DATA_BLOCK "A0301_Fermi_P2"   // DB36
// stored: InstanceOfName A0301_Fermi_P2_FB, InstanceOfType FB
"A0301_Fermi_P2_FB"
BEGIN
   AreaInterface.EStop := FALSE;
   AreaInterface.Man := TRUE;
   AreaInterface.Aut := FALSE;
   AreaInterface.Cycle := FALSE;
   AreaInterface.StopInPhase := FALSE;
   AreaInterface.StopProgrammed := FALSE;
   AreaInterface.RstAlarms := FALSE;
   AreaInterface.ManOneShot := FALSE;
   AreaInterface.AutOneShot := FALSE;
   AreaInterface.CycleOneShot := FALSE;
   AreaInterface.CheckAutReady := FALSE;
   ZSI.Door_NormalStop := FALSE;
   ZSI.Door_SafeStop := FALSE;
   ZSI.Door_Opened := FALSE;
   ZSI.Door_EntryEnable := FALSE;
   DSI.SafeStop := FALSE;
   DSI.PowerEnable := TRUE;
   DSI.DevicesInSafeState := FALSE;
   CIn.Manager_Fermi.EnableStopDoorOpeningReq := FALSE;
   CIn.Manager_Fermi.EnableStopInPhase := FALSE;
   CIn.Manager_Fermi.EnableStopProgrammed := FALSE;
   CIn.Manager_Fermi.Control_ON := FALSE;
   CIn.Manager_Fermi.Rest := FALSE;
   CIn.Manager_Fermi.Work := FALSE;
   CIn.P1.Fermi.CtrlSafe := FALSE;
   CIn.P1.Fermi.Standstill := TRUE;
   CIn.P1.Fermi.ReqOilPressure := FALSE;
   CIn.P1.Fermi.Rest_CheckNext := FALSE;
   CIn.P1.Fermi.Work_CheckNext := FALSE;
   CIn.P1.Fermi.Rest := FALSE;
   CIn.P1.Fermi.Work := FALSE;
   CIn.P1.Pareggiatore.CtrlSafe := FALSE;
   CIn.P1.Pareggiatore.Standstill := TRUE;
   CIn.P1.Pareggiatore.ReqOilPressure := FALSE;
   CIn.P1.Pareggiatore.Rest_CheckNext := FALSE;
   CIn.P1.Pareggiatore.Work_CheckNext := FALSE;
   CIn.P1.Pareggiatore.Rest := FALSE;
   CIn.P1.Pareggiatore.Work := FALSE;
   CIn.Trasporto.Infeed_ReqON := FALSE;
   CIn.Trasporto.CtrlSafe := FALSE;
   CIn.Trasporto.Standstill := TRUE;
   CIn.Trasporto.Bwd_CheckNext := FALSE;
   CIn.Trasporto.Fwd_CheckNext := FALSE;
   CIn.Trasporto.Bwd_VelZero := FALSE;
   CIn.Trasporto.Bwd_Running := FALSE;
   CIn.Trasporto.Fwd_VelZero := FALSE;
   CIn.Trasporto.Fwd_Running := FALSE;
   CIn.Trasporto.ActualVelocity := 0.0;
   CIn.Trasporto.TargetVelocity := 0.0;
   CIn.Trasporto.MaxVelocity := 39597.8;
   Config.Fermi[1..6].DelayPressureRunningTimeout := T#3S;
   Config.Fermi[1..6].DelayMissingCondition := T#3S;
   Config.Fermi[1..6].Rest_LsQty := 1;
   Config.Fermi[1..6].Work_LsQty := 0;
   Config.Fermi[1..6].Rest_RetainAut := FALSE;
   Config.Fermi[1..6].Work_RetainAut := FALSE;
   Config.Fermi[1..6].V.RestLimSwitchExist := TRUE;
   Config.Fermi[1..6].V.WorkLimSwitchExist := FALSE;
   Config.Fermi[1..6].V.CheckOilInPressure := FALSE;
   Config.Fermi[1..6].V.CutRestWhenIsAtRest := TRUE;
   Config.Fermi[1..6].V.CutWorkWhenIsAtWork := TRUE;
   Config.Fermi[1..6].V.RestTime := T#2S;
   Config.Fermi[1..6].V.WorkTime := T#2S;
   Config.Fermi[1..6].V.RestTimeOut := T#1H;
   Config.Fermi[1..6].V.WorkTimeOut := T#1H;
   Config.Sollevatori[1..6].DelayPressureRunningTimeout := T#3S;
   Config.Sollevatori[1..6].DelayMissingCondition := T#3S;
   Config.Sollevatori[1..6].Rest_LsQty := 1;
   Config.Sollevatori[1..6].Work_LsQty := 0;
   Config.Sollevatori[1..6].Rest_RetainAut := FALSE;
   Config.Sollevatori[1..6].Work_RetainAut := FALSE;
   Config.Sollevatori[1..6].V.RestLimSwitchExist := TRUE;
   Config.Sollevatori[1..6].V.WorkLimSwitchExist := FALSE;
   Config.Sollevatori[1..6].V.CheckOilInPressure := FALSE;
   Config.Sollevatori[1..6].V.CutRestWhenIsAtRest := TRUE;
   Config.Sollevatori[1..6].V.CutWorkWhenIsAtWork := TRUE;
   Config.Sollevatori[1..6].V.RestTime := T#2S;
   Config.Sollevatori[1..6].V.WorkTime := T#2S;
   Config.Sollevatori[1..6].V.RestTimeOut := T#1H;
   Config.Sollevatori[1..6].V.WorkTimeOut := T#1H;
   MachineInterface.AutReady := FALSE;
   MachineInterface.Aborting := FALSE;
   MachineInterface.AckStopInPhase := FALSE;
   MachineInterface.AckStopProgrammed := FALSE;
   MachineInterface.MotionsStandStill := TRUE;
   MachineInterface.AlarmsPresence := FALSE;
   MachineInterface.WarningPresence := FALSE;
   COut.Fermi.CtrlSafe := FALSE;
   COut.Fermi.Standstill := TRUE;
   COut.Fermi.ReqOilPressure := FALSE;
   COut.Fermi.Rest_CheckNext := FALSE;
   COut.Fermi.Work_CheckNext := FALSE;
   COut.Fermi.Rest := FALSE;
   COut.Fermi.Work := FALSE;
   COut.Sollevatori.CtrlSafe := FALSE;
   COut.Sollevatori.Standstill := TRUE;
   COut.Sollevatori.ReqOilPressure := FALSE;
   COut.Sollevatori.Rest_CheckNext := FALSE;
   COut.Sollevatori.Work_CheckNext := FALSE;
   COut.Sollevatori.Rest := FALSE;
   COut.Sollevatori.Work := FALSE;
   Alarm.Fermi[1..6].TimeOutRest := FALSE;
   Alarm.Fermi[1..6].TimeOutWork := FALSE;
   Alarm.Fermi[1..6].LimitSwitches := FALSE;
   Alarm.Sollevatori[1..6].TimeOutRest := FALSE;
   Alarm.Sollevatori[1..6].TimeOutWork := FALSE;
   Alarm.Sollevatori[1..6].LimitSwitches := FALSE;
   Warning.Fermi[1..6].NotAutReady := FALSE;
   Warning.Fermi[1..6].PressureRunning_Timeout := FALSE;
   Warning.Fermi[1..6].Rest_MissingExtEnable := FALSE;
   Warning.Fermi[1..6].Work_MissingExtEnable := FALSE;
   Warning.Fermi[1].Missing_Rest_Ls_ON[1..8] := FALSE;
   Warning.Fermi[2].Missing_Rest_Ls_ON[1..8] := FALSE;
   Warning.Fermi[3].Missing_Rest_Ls_ON[1..8] := FALSE;
   Warning.Fermi[4].Missing_Rest_Ls_ON[1..8] := FALSE;
   Warning.Fermi[5].Missing_Rest_Ls_ON[1..8] := FALSE;
   Warning.Fermi[6].Missing_Rest_Ls_ON[1..8] := FALSE;
   Warning.Fermi[1].Missing_Work_Ls_ON[1..8] := FALSE;
   Warning.Fermi[2].Missing_Work_Ls_ON[1..8] := FALSE;
   Warning.Fermi[3].Missing_Work_Ls_ON[1..8] := FALSE;
   Warning.Fermi[4].Missing_Work_Ls_ON[1..8] := FALSE;
   Warning.Fermi[5].Missing_Work_Ls_ON[1..8] := FALSE;
   Warning.Fermi[6].Missing_Work_Ls_ON[1..8] := FALSE;
   Warning.Sollevatori[1..6].NotAutReady := FALSE;
   Warning.Sollevatori[1..6].PressureRunning_Timeout := FALSE;
   Warning.Sollevatori[1..6].Rest_MissingExtEnable := FALSE;
   Warning.Sollevatori[1..6].Work_MissingExtEnable := FALSE;
   Warning.Sollevatori[1].Missing_Rest_Ls_ON[1..8] := FALSE;
   Warning.Sollevatori[2].Missing_Rest_Ls_ON[1..8] := FALSE;
   Warning.Sollevatori[3].Missing_Rest_Ls_ON[1..8] := FALSE;
   Warning.Sollevatori[4].Missing_Rest_Ls_ON[1..8] := FALSE;
   Warning.Sollevatori[5].Missing_Rest_Ls_ON[1..8] := FALSE;
   Warning.Sollevatori[6].Missing_Rest_Ls_ON[1..8] := FALSE;
   Warning.Sollevatori[1].Missing_Work_Ls_ON[1..8] := FALSE;
   Warning.Sollevatori[2].Missing_Work_Ls_ON[1..8] := FALSE;
   Warning.Sollevatori[3].Missing_Work_Ls_ON[1..8] := FALSE;
   Warning.Sollevatori[4].Missing_Work_Ls_ON[1..8] := FALSE;
   Warning.Sollevatori[5].Missing_Work_Ls_ON[1..8] := FALSE;
   Warning.Sollevatori[6].Missing_Work_Ls_ON[1..8] := FALSE;
   HMI.Selection[1..6] := TRUE;
   HMI.FermiSts.Standstill := TRUE;
   HMI.FermiSts.Rest := FALSE;
   HMI.FermiSts.Work := FALSE;
   HMI.FermiSts.AlarmPresence := FALSE;
   HMI.SollevatoriSts.Standstill := TRUE;
   HMI.SollevatoriSts.Rest := FALSE;
   HMI.SollevatoriSts.Work := FALSE;
   HMI.SollevatoriSts.AlarmPresence := FALSE;
   Fermi[1..6].AreaInterface.EStop := FALSE;
   Fermi[1..6].AreaInterface.Man := TRUE;
   Fermi[1..6].AreaInterface.Aut := FALSE;
   Fermi[1..6].AreaInterface.Cycle := FALSE;
   Fermi[1..6].AreaInterface.StopInPhase := FALSE;
   Fermi[1..6].AreaInterface.StopProgrammed := FALSE;
   Fermi[1..6].AreaInterface.RstAlarms := FALSE;
   Fermi[1..6].AreaInterface.ManOneShot := FALSE;
   Fermi[1..6].AreaInterface.AutOneShot := FALSE;
   Fermi[1..6].AreaInterface.CycleOneShot := FALSE;
   Fermi[1..6].AreaInterface.CheckAutReady := FALSE;
   Fermi[1..6].ZSI.Door_NormalStop := FALSE;
   Fermi[1..6].ZSI.Door_SafeStop := FALSE;
   Fermi[1..6].ZSI.Door_Opened := FALSE;
   Fermi[1..6].ZSI.Door_EntryEnable := FALSE;
   Fermi[1..6].DSI.SafeStop := FALSE;
   Fermi[1..6].DSI.PowerEnable := TRUE;
   Fermi[1..6].DSI.DevicesInSafeState := FALSE;
   Fermi[1..6].DataIn.PB.Rest := FALSE;
   Fermi[1..6].DataIn.PB.Work := FALSE;
   Fermi[1..6].DataIn.PB.StartStop := FALSE;
   Fermi[1].DataIn.Rest_Ls[1] := TRUE;
   Fermi[1].DataIn.Rest_Ls[2..8] := FALSE;
   Fermi[2].DataIn.Rest_Ls[1] := TRUE;
   Fermi[2].DataIn.Rest_Ls[2..8] := FALSE;
   Fermi[3].DataIn.Rest_Ls[1] := TRUE;
   Fermi[3].DataIn.Rest_Ls[2..8] := FALSE;
   Fermi[4].DataIn.Rest_Ls[1] := TRUE;
   Fermi[4].DataIn.Rest_Ls[2..8] := FALSE;
   Fermi[5].DataIn.Rest_Ls[1] := TRUE;
   Fermi[5].DataIn.Rest_Ls[2..8] := FALSE;
   Fermi[6].DataIn.Rest_Ls[1] := TRUE;
   Fermi[6].DataIn.Rest_Ls[2..8] := FALSE;
   Fermi[1].DataIn.Work_Ls[1..8] := FALSE;
   Fermi[2].DataIn.Work_Ls[1..8] := FALSE;
   Fermi[3].DataIn.Work_Ls[1..8] := FALSE;
   Fermi[4].DataIn.Work_Ls[1..8] := FALSE;
   Fermi[5].DataIn.Work_Ls[1..8] := FALSE;
   Fermi[6].DataIn.Work_Ls[1..8] := FALSE;
   Fermi[1..6].Cin.Manager.EnableStopDoorOpeningReq := FALSE;
   Fermi[1..6].Cin.Manager.EnableStopInPhase := FALSE;
   Fermi[1..6].Cin.Manager.EnableStopProgrammed := FALSE;
   Fermi[1..6].Cin.Manager.Control_ON := FALSE;
   Fermi[1..6].Cin.Manager.Rest := FALSE;
   Fermi[1..6].Cin.Manager.Work := FALSE;
   Fermi[1..6].Cin.PressureRunning := FALSE;
   Fermi[1..6].Cin.Rest_ExtEnable := TRUE;
   Fermi[1..6].Cin.Work_ExtEnable := TRUE;
   Fermi[1..6].Cin.ExternalAlarms := FALSE;
   Fermi[1..6].Config.DelayPressureRunningTimeout := T#3S;
   Fermi[1..6].Config.DelayMissingCondition := T#3S;
   Fermi[1..6].Config.Rest_LsQty := 1;
   Fermi[1..6].Config.Work_LsQty := 0;
   Fermi[1..6].Config.Rest_RetainAut := FALSE;
   Fermi[1..6].Config.Work_RetainAut := FALSE;
   Fermi[1..6].Config.V.RestLimSwitchExist := TRUE;
   Fermi[1..6].Config.V.WorkLimSwitchExist := FALSE;
   Fermi[1..6].Config.V.CheckOilInPressure := FALSE;
   Fermi[1..6].Config.V.CutRestWhenIsAtRest := TRUE;
   Fermi[1..6].Config.V.CutWorkWhenIsAtWork := TRUE;
   Fermi[1..6].Config.V.RestTime := T#2S;
   Fermi[1..6].Config.V.WorkTime := T#2S;
   Fermi[1..6].Config.V.RestTimeOut := T#1H;
   Fermi[1..6].Config.V.WorkTimeOut := T#1H;
   Fermi[1..6].MachineInterface.AutReady := FALSE;
   Fermi[1..6].MachineInterface.Aborting := FALSE;
   Fermi[1..6].MachineInterface.AckStopInPhase := FALSE;
   Fermi[1..6].MachineInterface.AckStopProgrammed := FALSE;
   Fermi[1..6].MachineInterface.MotionsStandStill := TRUE;
   Fermi[1..6].MachineInterface.AlarmsPresence := FALSE;
   Fermi[1..6].MachineInterface.WarningPresence := FALSE;
   Fermi[1..6].COut.CtrlSafe := FALSE;
   Fermi[1..6].COut.Standstill := TRUE;
   Fermi[1..6].COut.ReqOilPressure := FALSE;
   Fermi[1..6].COut.Rest_CheckNext := FALSE;
   Fermi[1..6].COut.Work_CheckNext := FALSE;
   Fermi[1..6].COut.Rest := TRUE;
   Fermi[1..6].COut.Work := FALSE;
   Fermi[1..6].DataOut.RestSolenoid := FALSE;
   Fermi[1..6].DataOut.WorkSolenoid := FALSE;
   Fermi[1..6].Sts.Standstill := TRUE;
   Fermi[1..6].Sts.AlarmsPresence := FALSE;
   Fermi[1..6].Sts.WarningsPresence := FALSE;
   Fermi[1..6].Sts.Rest_Cnd := TRUE;
   Fermi[1..6].Sts.Work_Cnd := TRUE;
   Fermi[1..6].Ctrl.StopDueDoorOpeningRequest := FALSE;
   Fermi[1..6].Ctrl.StopInPhase := FALSE;
   Fermi[1..6].Ctrl.StopProgrammed := FALSE;
   Fermi[1..6].Ctrl.StopAborting := FALSE;
   Fermi[1..6].Ctrl.Work := FALSE;
   Fermi[1..6].Ctrl.Rest := FALSE;
   Fermi[1..6].Ctrl.Rest_Man := FALSE;
   Fermi[1..6].Ctrl.Work_Man := FALSE;
   Fermi[1..6].Ctrl.Rest_Aut := FALSE;
   Fermi[1..6].Ctrl.Work_Aut := FALSE;
   Fermi[1..6].V.ValveCtrl.SafeStop := FALSE;
   Fermi[1..6].V.ValveCtrl.Rst := FALSE;
   Fermi[1..6].V.ValveCtrl.MoveRest := FALSE;
   Fermi[1..6].V.ValveCtrl.MoveWork := FALSE;
   Fermi[1..6].V.RestLimitSwitch := TRUE;
   Fermi[1..6].V.WorkLimitSwitch := FALSE;
   Fermi[1..6].V.OilInPressure := FALSE;
   Fermi[1..6].V.Simulation := FALSE;
   Fermi[1..6].V.Config.RestLimSwitchExist := TRUE;
   Fermi[1..6].V.Config.WorkLimSwitchExist := FALSE;
   Fermi[1..6].V.Config.CheckOilInPressure := FALSE;
   Fermi[1..6].V.Config.CutRestWhenIsAtRest := TRUE;
   Fermi[1..6].V.Config.CutWorkWhenIsAtWork := TRUE;
   Fermi[1..6].V.Config.RestTime := T#2S;
   Fermi[1..6].V.Config.WorkTime := T#2S;
   Fermi[1..6].V.Config.RestTimeOut := T#1H;
   Fermi[1..6].V.Config.WorkTimeOut := T#1H;
   Fermi[1..6].V.ValveSts.AlarmPresence := FALSE;
   Fermi[1..6].V.ValveSts.RestPermit := TRUE;
   Fermi[1..6].V.ValveSts.RestInProgress := FALSE;
   Fermi[1..6].V.ValveSts.IsAtRest := TRUE;
   Fermi[1..6].V.ValveSts.WorkPermit := TRUE;
   Fermi[1..6].V.ValveSts.WorkInProgress := FALSE;
   Fermi[1..6].V.ValveSts.IsAtWork := FALSE;
   Fermi[1..6].V.ValveSts.StandStill := TRUE;
   Fermi[1..6].V.RestSolenoid := FALSE;
   Fermi[1..6].V.WorkSolenoid := FALSE;
   Fermi[1..6].V.ReqOilPressure := FALSE;
   Fermi[1..6].V.IsAtRest := TRUE;
   Fermi[1..6].V.IsAtWork := FALSE;
   Fermi[1..6].V.Ctrl.RestReq := FALSE;
   Fermi[1..6].V.Ctrl.WorkReq := FALSE;
   Fermi[1..6].V.Ctrl.RestSolenoid := FALSE;
   Fermi[1..6].V.Ctrl.WorkSolenoid := FALSE;
   Fermi[1..6].V.tonRest.PT := T#2S;
   Fermi[1..6].V.tonRest.IN := TRUE;
   Fermi[1..6].V.tonWork.PT := T#0MS;
   Fermi[1..6].V.tonWork.IN := FALSE;
   Fermi[1..6].V.tonTimeOutRest.PT := T#0MS;
   Fermi[1..6].V.tonTimeOutRest.IN := FALSE;
   Fermi[1..6].V.tonTimeOutWork.PT := T#0MS;
   Fermi[1..6].V.tonTimeOutWork.IN := FALSE;
   Fermi[1..6].TON_NoPendingCmd.PT := T#500MS;
   Fermi[1..6].TON_NoPendingCmd.IN := TRUE;
   Fermi[1..6].TON_Rest_MissingExtEnable.PT := T#0MS;
   Fermi[1..6].TON_Rest_MissingExtEnable.IN := FALSE;
   Fermi[1..6].TON_Work_MissingExtEnable.PT := T#0MS;
   Fermi[1..6].TON_Work_MissingExtEnable.IN := FALSE;
   Fermi[1..6].TON_PressureRunning_Timeout.PT := T#0MS;
   Fermi[1..6].TON_PressureRunning_Timeout.IN := FALSE;
   Fermi[1..6].Aux.Pb_Rest := FALSE;
   Fermi[1..6].Aux.Pb_Work := FALSE;
   Fermi[1..6].Aux.Pb_StartStop := FALSE;
   Sollevatori[1..6].AreaInterface.EStop := FALSE;
   Sollevatori[1..6].AreaInterface.Man := TRUE;
   Sollevatori[1..6].AreaInterface.Aut := FALSE;
   Sollevatori[1..6].AreaInterface.Cycle := FALSE;
   Sollevatori[1..6].AreaInterface.StopInPhase := FALSE;
   Sollevatori[1..6].AreaInterface.StopProgrammed := FALSE;
   Sollevatori[1..6].AreaInterface.RstAlarms := FALSE;
   Sollevatori[1..6].AreaInterface.ManOneShot := FALSE;
   Sollevatori[1..6].AreaInterface.AutOneShot := FALSE;
   Sollevatori[1..6].AreaInterface.CycleOneShot := FALSE;
   Sollevatori[1..6].AreaInterface.CheckAutReady := FALSE;
   Sollevatori[1..6].ZSI.Door_NormalStop := FALSE;
   Sollevatori[1..6].ZSI.Door_SafeStop := FALSE;
   Sollevatori[1..6].ZSI.Door_Opened := FALSE;
   Sollevatori[1..6].ZSI.Door_EntryEnable := FALSE;
   Sollevatori[1..6].DSI.SafeStop := FALSE;
   Sollevatori[1..6].DSI.PowerEnable := TRUE;
   Sollevatori[1..6].DSI.DevicesInSafeState := FALSE;
   Sollevatori[1..6].DataIn.PB.Rest := FALSE;
   Sollevatori[1..6].DataIn.PB.Work := FALSE;
   Sollevatori[1..6].DataIn.PB.StartStop := FALSE;
   Sollevatori[1].DataIn.Rest_Ls[1] := TRUE;
   Sollevatori[1].DataIn.Rest_Ls[2..8] := FALSE;
   Sollevatori[2].DataIn.Rest_Ls[1] := TRUE;
   Sollevatori[2].DataIn.Rest_Ls[2..8] := FALSE;
   Sollevatori[3].DataIn.Rest_Ls[1] := TRUE;
   Sollevatori[3].DataIn.Rest_Ls[2..8] := FALSE;
   Sollevatori[4].DataIn.Rest_Ls[1] := TRUE;
   Sollevatori[4].DataIn.Rest_Ls[2..8] := FALSE;
   Sollevatori[5].DataIn.Rest_Ls[1] := TRUE;
   Sollevatori[5].DataIn.Rest_Ls[2..8] := FALSE;
   Sollevatori[6].DataIn.Rest_Ls[1] := TRUE;
   Sollevatori[6].DataIn.Rest_Ls[2..8] := FALSE;
   Sollevatori[1].DataIn.Work_Ls[1..8] := FALSE;
   Sollevatori[2].DataIn.Work_Ls[1..8] := FALSE;
   Sollevatori[3].DataIn.Work_Ls[1..8] := FALSE;
   Sollevatori[4].DataIn.Work_Ls[1..8] := FALSE;
   Sollevatori[5].DataIn.Work_Ls[1..8] := FALSE;
   Sollevatori[6].DataIn.Work_Ls[1..8] := FALSE;
   Sollevatori[1..6].Cin.Manager.EnableStopDoorOpeningReq := FALSE;
   Sollevatori[1..6].Cin.Manager.EnableStopInPhase := FALSE;
   Sollevatori[1..6].Cin.Manager.EnableStopProgrammed := FALSE;
   Sollevatori[1..6].Cin.Manager.Control_ON := FALSE;
   Sollevatori[1..6].Cin.Manager.Rest := FALSE;
   Sollevatori[1..6].Cin.Manager.Work := FALSE;
   Sollevatori[1..6].Cin.PressureRunning := FALSE;
   Sollevatori[1..6].Cin.Rest_ExtEnable := TRUE;
   Sollevatori[1..6].Cin.Work_ExtEnable := TRUE;
   Sollevatori[1..6].Cin.ExternalAlarms := FALSE;
   Sollevatori[1..6].Config.DelayPressureRunningTimeout := T#3S;
   Sollevatori[1..6].Config.DelayMissingCondition := T#3S;
   Sollevatori[1..6].Config.Rest_LsQty := 1;
   Sollevatori[1..6].Config.Work_LsQty := 0;
   Sollevatori[1..6].Config.Rest_RetainAut := FALSE;
   Sollevatori[1..6].Config.Work_RetainAut := FALSE;
   Sollevatori[1..6].Config.V.RestLimSwitchExist := TRUE;
   Sollevatori[1..6].Config.V.WorkLimSwitchExist := FALSE;
   Sollevatori[1..6].Config.V.CheckOilInPressure := FALSE;
   Sollevatori[1..6].Config.V.CutRestWhenIsAtRest := TRUE;
   Sollevatori[1..6].Config.V.CutWorkWhenIsAtWork := TRUE;
   Sollevatori[1..6].Config.V.RestTime := T#2S;
   Sollevatori[1..6].Config.V.WorkTime := T#2S;
   Sollevatori[1..6].Config.V.RestTimeOut := T#1H;
   Sollevatori[1..6].Config.V.WorkTimeOut := T#1H;
   Sollevatori[1..6].MachineInterface.AutReady := FALSE;
   Sollevatori[1..6].MachineInterface.Aborting := FALSE;
   Sollevatori[1..6].MachineInterface.AckStopInPhase := FALSE;
   Sollevatori[1..6].MachineInterface.AckStopProgrammed := FALSE;
   Sollevatori[1..6].MachineInterface.MotionsStandStill := TRUE;
   Sollevatori[1..6].MachineInterface.AlarmsPresence := FALSE;
   Sollevatori[1..6].MachineInterface.WarningPresence := FALSE;
   Sollevatori[1..6].COut.CtrlSafe := FALSE;
   Sollevatori[1..6].COut.Standstill := TRUE;
   Sollevatori[1..6].COut.ReqOilPressure := FALSE;
   Sollevatori[1..6].COut.Rest_CheckNext := FALSE;
   Sollevatori[1..6].COut.Work_CheckNext := FALSE;
   Sollevatori[1..6].COut.Rest := TRUE;
   Sollevatori[1..6].COut.Work := FALSE;
   Sollevatori[1..6].DataOut.RestSolenoid := FALSE;
   Sollevatori[1..6].DataOut.WorkSolenoid := FALSE;
   Sollevatori[1..6].Sts.Standstill := TRUE;
   Sollevatori[1..6].Sts.AlarmsPresence := FALSE;
   Sollevatori[1..6].Sts.WarningsPresence := FALSE;
   Sollevatori[1..6].Sts.Rest_Cnd := TRUE;
   Sollevatori[1..6].Sts.Work_Cnd := TRUE;
   Sollevatori[1..6].Ctrl.StopDueDoorOpeningRequest := FALSE;
   Sollevatori[1..6].Ctrl.StopInPhase := FALSE;
   Sollevatori[1..6].Ctrl.StopProgrammed := FALSE;
   Sollevatori[1..6].Ctrl.StopAborting := FALSE;
   Sollevatori[1..6].Ctrl.Work := FALSE;
   Sollevatori[1..6].Ctrl.Rest := FALSE;
   Sollevatori[1..6].Ctrl.Rest_Man := FALSE;
   Sollevatori[1..6].Ctrl.Work_Man := FALSE;
   Sollevatori[1..6].Ctrl.Rest_Aut := FALSE;
   Sollevatori[1..6].Ctrl.Work_Aut := FALSE;
   Sollevatori[1..6].V.ValveCtrl.SafeStop := FALSE;
   Sollevatori[1..6].V.ValveCtrl.Rst := FALSE;
   Sollevatori[1..6].V.ValveCtrl.MoveRest := FALSE;
   Sollevatori[1..6].V.ValveCtrl.MoveWork := FALSE;
   Sollevatori[1..6].V.RestLimitSwitch := TRUE;
   Sollevatori[1..6].V.WorkLimitSwitch := FALSE;
   Sollevatori[1..6].V.OilInPressure := FALSE;
   Sollevatori[1..6].V.Simulation := FALSE;
   Sollevatori[1..6].V.Config.RestLimSwitchExist := TRUE;
   Sollevatori[1..6].V.Config.WorkLimSwitchExist := FALSE;
   Sollevatori[1..6].V.Config.CheckOilInPressure := FALSE;
   Sollevatori[1..6].V.Config.CutRestWhenIsAtRest := TRUE;
   Sollevatori[1..6].V.Config.CutWorkWhenIsAtWork := TRUE;
   Sollevatori[1..6].V.Config.RestTime := T#2S;
   Sollevatori[1..6].V.Config.WorkTime := T#2S;
   Sollevatori[1..6].V.Config.RestTimeOut := T#1H;
   Sollevatori[1..6].V.Config.WorkTimeOut := T#1H;
   Sollevatori[1..6].V.ValveSts.AlarmPresence := FALSE;
   Sollevatori[1..6].V.ValveSts.RestPermit := TRUE;
   Sollevatori[1..6].V.ValveSts.RestInProgress := FALSE;
   Sollevatori[1..6].V.ValveSts.IsAtRest := TRUE;
   Sollevatori[1..6].V.ValveSts.WorkPermit := TRUE;
   Sollevatori[1..6].V.ValveSts.WorkInProgress := FALSE;
   Sollevatori[1..6].V.ValveSts.IsAtWork := FALSE;
   Sollevatori[1..6].V.ValveSts.StandStill := TRUE;
   Sollevatori[1..6].V.RestSolenoid := FALSE;
   Sollevatori[1..6].V.WorkSolenoid := FALSE;
   Sollevatori[1..6].V.ReqOilPressure := FALSE;
   Sollevatori[1..6].V.IsAtRest := TRUE;
   Sollevatori[1..6].V.IsAtWork := FALSE;
   Sollevatori[1..6].V.Ctrl.RestReq := FALSE;
   Sollevatori[1..6].V.Ctrl.WorkReq := FALSE;
   Sollevatori[1..6].V.Ctrl.RestSolenoid := FALSE;
   Sollevatori[1..6].V.Ctrl.WorkSolenoid := FALSE;
   Sollevatori[1..6].V.tonRest.PT := T#2S;
   Sollevatori[1..6].V.tonRest.IN := TRUE;
   Sollevatori[1..6].V.tonWork.PT := T#0MS;
   Sollevatori[1..6].V.tonWork.IN := FALSE;
   Sollevatori[1..6].V.tonTimeOutRest.PT := T#0MS;
   Sollevatori[1..6].V.tonTimeOutRest.IN := FALSE;
   Sollevatori[1..6].V.tonTimeOutWork.PT := T#0MS;
   Sollevatori[1..6].V.tonTimeOutWork.IN := FALSE;
   Sollevatori[1..6].TON_NoPendingCmd.PT := T#500MS;
   Sollevatori[1..6].TON_NoPendingCmd.IN := TRUE;
   Sollevatori[1..6].TON_Rest_MissingExtEnable.PT := T#0MS;
   Sollevatori[1..6].TON_Rest_MissingExtEnable.IN := FALSE;
   Sollevatori[1..6].TON_Work_MissingExtEnable.PT := T#0MS;
   Sollevatori[1..6].TON_Work_MissingExtEnable.IN := FALSE;
   Sollevatori[1..6].TON_PressureRunning_Timeout.PT := T#0MS;
   Sollevatori[1..6].TON_PressureRunning_Timeout.IN := FALSE;
   Sollevatori[1..6].Aux.Pb_Rest := FALSE;
   Sollevatori[1..6].Aux.Pb_Work := FALSE;
   Sollevatori[1..6].Aux.Pb_StartStop := FALSE;
   TON_OP_REST_MissingCnd.PT := T#0MS;
   TON_OP_REST_MissingCnd.IN := FALSE;
   TON_OP_WORK_MissingCnd.PT := T#0MS;
   TON_OP_WORK_MissingCnd.IN := FALSE;
END_DATA_BLOCK

DATA_BLOCK "A0301_Fermi_P3"   // DB56
// stored: InstanceOfName A0301_Fermi_P3_FB, InstanceOfType FB
"A0301_Fermi_P3_FB"
BEGIN
   AreaInterface.EStop := FALSE;
   AreaInterface.Man := TRUE;
   AreaInterface.Aut := FALSE;
   AreaInterface.Cycle := FALSE;
   AreaInterface.StopInPhase := FALSE;
   AreaInterface.StopProgrammed := FALSE;
   AreaInterface.RstAlarms := FALSE;
   AreaInterface.ManOneShot := FALSE;
   AreaInterface.AutOneShot := FALSE;
   AreaInterface.CycleOneShot := FALSE;
   AreaInterface.CheckAutReady := FALSE;
   ZSI.Door_NormalStop := FALSE;
   ZSI.Door_SafeStop := FALSE;
   ZSI.Door_Opened := FALSE;
   ZSI.Door_EntryEnable := FALSE;
   DSI.SafeStop := FALSE;
   DSI.PowerEnable := TRUE;
   DSI.DevicesInSafeState := FALSE;
   CIn.Manager.EnableStopDoorOpeningReq := FALSE;
   CIn.Manager.EnableStopInPhase := FALSE;
   CIn.Manager.EnableStopProgrammed := FALSE;
   CIn.Manager.Control_ON := FALSE;
   CIn.Manager.Rest := FALSE;
   CIn.Manager.Work := FALSE;
   CIn.P2.Fermi.CtrlSafe := FALSE;
   CIn.P2.Fermi.Standstill := TRUE;
   CIn.P2.Fermi.ReqOilPressure := FALSE;
   CIn.P2.Fermi.Rest_CheckNext := FALSE;
   CIn.P2.Fermi.Work_CheckNext := FALSE;
   CIn.P2.Fermi.Rest := FALSE;
   CIn.P2.Fermi.Work := FALSE;
   CIn.P2.Sollevatore.CtrlSafe := FALSE;
   CIn.P2.Sollevatore.Standstill := TRUE;
   CIn.P2.Sollevatore.ReqOilPressure := FALSE;
   CIn.P2.Sollevatore.Rest_CheckNext := FALSE;
   CIn.P2.Sollevatore.Work_CheckNext := FALSE;
   CIn.P2.Sollevatore.Rest := FALSE;
   CIn.P2.Sollevatore.Work := FALSE;
   CIn.Trasporto.Infeed_ReqON := FALSE;
   CIn.Trasporto.CtrlSafe := FALSE;
   CIn.Trasporto.Standstill := TRUE;
   CIn.Trasporto.Bwd_CheckNext := FALSE;
   CIn.Trasporto.Fwd_CheckNext := FALSE;
   CIn.Trasporto.Bwd_VelZero := FALSE;
   CIn.Trasporto.Bwd_Running := FALSE;
   CIn.Trasporto.Fwd_VelZero := FALSE;
   CIn.Trasporto.Fwd_Running := FALSE;
   CIn.Trasporto.ActualVelocity := 0.0;
   CIn.Trasporto.TargetVelocity := 0.0;
   CIn.Trasporto.MaxVelocity := 39597.8;
   Config.Fermi[1..6].DelayPressureRunningTimeout := T#3S;
   Config.Fermi[1..6].DelayMissingCondition := T#3S;
   Config.Fermi[1..6].Rest_LsQty := 1;
   Config.Fermi[1..6].Work_LsQty := 0;
   Config.Fermi[1..6].Rest_RetainAut := FALSE;
   Config.Fermi[1..6].Work_RetainAut := FALSE;
   Config.Fermi[1..6].V.RestLimSwitchExist := TRUE;
   Config.Fermi[1..6].V.WorkLimSwitchExist := FALSE;
   Config.Fermi[1..6].V.CheckOilInPressure := FALSE;
   Config.Fermi[1..6].V.CutRestWhenIsAtRest := TRUE;
   Config.Fermi[1..6].V.CutWorkWhenIsAtWork := TRUE;
   Config.Fermi[1..6].V.RestTime := T#2S;
   Config.Fermi[1..6].V.WorkTime := T#2S;
   Config.Fermi[1..6].V.RestTimeOut := T#1H;
   Config.Fermi[1..6].V.WorkTimeOut := T#1H;
   MachineInterface.AutReady := FALSE;
   MachineInterface.Aborting := FALSE;
   MachineInterface.AckStopInPhase := FALSE;
   MachineInterface.AckStopProgrammed := FALSE;
   MachineInterface.MotionsStandStill := TRUE;
   MachineInterface.AlarmsPresence := FALSE;
   MachineInterface.WarningPresence := FALSE;
   COut.Fermi.CtrlSafe := FALSE;
   COut.Fermi.Standstill := TRUE;
   COut.Fermi.ReqOilPressure := FALSE;
   COut.Fermi.Rest_CheckNext := FALSE;
   COut.Fermi.Work_CheckNext := FALSE;
   COut.Fermi.Rest := FALSE;
   COut.Fermi.Work := FALSE;
   Alarm.Fermi[1..6].TimeOutRest := FALSE;
   Alarm.Fermi[1..6].TimeOutWork := FALSE;
   Alarm.Fermi[1..6].LimitSwitches := FALSE;
   Warning.Fermi[1..6].NotAutReady := FALSE;
   Warning.Fermi[1..6].PressureRunning_Timeout := FALSE;
   Warning.Fermi[1..6].Rest_MissingExtEnable := FALSE;
   Warning.Fermi[1..6].Work_MissingExtEnable := FALSE;
   Warning.Fermi[1].Missing_Rest_Ls_ON[1..8] := FALSE;
   Warning.Fermi[2].Missing_Rest_Ls_ON[1..8] := FALSE;
   Warning.Fermi[3].Missing_Rest_Ls_ON[1..8] := FALSE;
   Warning.Fermi[4].Missing_Rest_Ls_ON[1..8] := FALSE;
   Warning.Fermi[5].Missing_Rest_Ls_ON[1..8] := FALSE;
   Warning.Fermi[6].Missing_Rest_Ls_ON[1..8] := FALSE;
   Warning.Fermi[1].Missing_Work_Ls_ON[1..8] := FALSE;
   Warning.Fermi[2].Missing_Work_Ls_ON[1..8] := FALSE;
   Warning.Fermi[3].Missing_Work_Ls_ON[1..8] := FALSE;
   Warning.Fermi[4].Missing_Work_Ls_ON[1..8] := FALSE;
   Warning.Fermi[5].Missing_Work_Ls_ON[1..8] := FALSE;
   Warning.Fermi[6].Missing_Work_Ls_ON[1..8] := FALSE;
   HMI.Selection[1..6] := TRUE;
   HMI.FermiSts.Standstill := TRUE;
   HMI.FermiSts.Rest := FALSE;
   HMI.FermiSts.Work := FALSE;
   HMI.FermiSts.AlarmPresence := FALSE;
   Fermi[1..6].AreaInterface.EStop := FALSE;
   Fermi[1..6].AreaInterface.Man := TRUE;
   Fermi[1..6].AreaInterface.Aut := FALSE;
   Fermi[1..6].AreaInterface.Cycle := FALSE;
   Fermi[1..6].AreaInterface.StopInPhase := FALSE;
   Fermi[1..6].AreaInterface.StopProgrammed := FALSE;
   Fermi[1..6].AreaInterface.RstAlarms := FALSE;
   Fermi[1..6].AreaInterface.ManOneShot := FALSE;
   Fermi[1..6].AreaInterface.AutOneShot := FALSE;
   Fermi[1..6].AreaInterface.CycleOneShot := FALSE;
   Fermi[1..6].AreaInterface.CheckAutReady := FALSE;
   Fermi[1..6].ZSI.Door_NormalStop := FALSE;
   Fermi[1..6].ZSI.Door_SafeStop := FALSE;
   Fermi[1..6].ZSI.Door_Opened := FALSE;
   Fermi[1..6].ZSI.Door_EntryEnable := FALSE;
   Fermi[1..6].DSI.SafeStop := FALSE;
   Fermi[1..6].DSI.PowerEnable := TRUE;
   Fermi[1..6].DSI.DevicesInSafeState := FALSE;
   Fermi[1..6].DataIn.PB.Rest := FALSE;
   Fermi[1..6].DataIn.PB.Work := FALSE;
   Fermi[1..6].DataIn.PB.StartStop := FALSE;
   Fermi[1].DataIn.Rest_Ls[1] := TRUE;
   Fermi[1].DataIn.Rest_Ls[2..8] := FALSE;
   Fermi[2].DataIn.Rest_Ls[1] := TRUE;
   Fermi[2].DataIn.Rest_Ls[2..8] := FALSE;
   Fermi[3].DataIn.Rest_Ls[1] := TRUE;
   Fermi[3].DataIn.Rest_Ls[2..8] := FALSE;
   Fermi[4].DataIn.Rest_Ls[1] := TRUE;
   Fermi[4].DataIn.Rest_Ls[2..8] := FALSE;
   Fermi[5].DataIn.Rest_Ls[1] := TRUE;
   Fermi[5].DataIn.Rest_Ls[2..8] := FALSE;
   Fermi[6].DataIn.Rest_Ls[1] := TRUE;
   Fermi[6].DataIn.Rest_Ls[2..8] := FALSE;
   Fermi[1].DataIn.Work_Ls[1..8] := FALSE;
   Fermi[2].DataIn.Work_Ls[1..8] := FALSE;
   Fermi[3].DataIn.Work_Ls[1..8] := FALSE;
   Fermi[4].DataIn.Work_Ls[1..8] := FALSE;
   Fermi[5].DataIn.Work_Ls[1..8] := FALSE;
   Fermi[6].DataIn.Work_Ls[1..8] := FALSE;
   Fermi[1..6].Cin.Manager.EnableStopDoorOpeningReq := FALSE;
   Fermi[1..6].Cin.Manager.EnableStopInPhase := FALSE;
   Fermi[1..6].Cin.Manager.EnableStopProgrammed := FALSE;
   Fermi[1..6].Cin.Manager.Control_ON := FALSE;
   Fermi[1..6].Cin.Manager.Rest := FALSE;
   Fermi[1..6].Cin.Manager.Work := FALSE;
   Fermi[1..6].Cin.PressureRunning := FALSE;
   Fermi[1..6].Cin.Rest_ExtEnable := TRUE;
   Fermi[1..6].Cin.Work_ExtEnable := TRUE;
   Fermi[1..6].Cin.ExternalAlarms := FALSE;
   Fermi[1..6].Config.DelayPressureRunningTimeout := T#3S;
   Fermi[1..6].Config.DelayMissingCondition := T#3S;
   Fermi[1..6].Config.Rest_LsQty := 1;
   Fermi[1..6].Config.Work_LsQty := 0;
   Fermi[1..6].Config.Rest_RetainAut := FALSE;
   Fermi[1..6].Config.Work_RetainAut := FALSE;
   Fermi[1..6].Config.V.RestLimSwitchExist := TRUE;
   Fermi[1..6].Config.V.WorkLimSwitchExist := FALSE;
   Fermi[1..6].Config.V.CheckOilInPressure := FALSE;
   Fermi[1..6].Config.V.CutRestWhenIsAtRest := TRUE;
   Fermi[1..6].Config.V.CutWorkWhenIsAtWork := TRUE;
   Fermi[1..6].Config.V.RestTime := T#2S;
   Fermi[1..6].Config.V.WorkTime := T#2S;
   Fermi[1..6].Config.V.RestTimeOut := T#1H;
   Fermi[1..6].Config.V.WorkTimeOut := T#1H;
   Fermi[1..6].MachineInterface.AutReady := FALSE;
   Fermi[1..6].MachineInterface.Aborting := FALSE;
   Fermi[1..6].MachineInterface.AckStopInPhase := FALSE;
   Fermi[1..6].MachineInterface.AckStopProgrammed := FALSE;
   Fermi[1..6].MachineInterface.MotionsStandStill := TRUE;
   Fermi[1..6].MachineInterface.AlarmsPresence := FALSE;
   Fermi[1..6].MachineInterface.WarningPresence := FALSE;
   Fermi[1..6].COut.CtrlSafe := FALSE;
   Fermi[1..6].COut.Standstill := TRUE;
   Fermi[1..6].COut.ReqOilPressure := FALSE;
   Fermi[1..6].COut.Rest_CheckNext := FALSE;
   Fermi[1..6].COut.Work_CheckNext := FALSE;
   Fermi[1..6].COut.Rest := TRUE;
   Fermi[1..6].COut.Work := FALSE;
   Fermi[1..6].DataOut.RestSolenoid := FALSE;
   Fermi[1..6].DataOut.WorkSolenoid := FALSE;
   Fermi[1..6].Sts.Standstill := TRUE;
   Fermi[1..6].Sts.AlarmsPresence := FALSE;
   Fermi[1..6].Sts.WarningsPresence := FALSE;
   Fermi[1..6].Sts.Rest_Cnd := TRUE;
   Fermi[1..6].Sts.Work_Cnd := TRUE;
   Fermi[1..6].Ctrl.StopDueDoorOpeningRequest := FALSE;
   Fermi[1..6].Ctrl.StopInPhase := FALSE;
   Fermi[1..6].Ctrl.StopProgrammed := FALSE;
   Fermi[1..6].Ctrl.StopAborting := FALSE;
   Fermi[1..6].Ctrl.Work := FALSE;
   Fermi[1..6].Ctrl.Rest := FALSE;
   Fermi[1..6].Ctrl.Rest_Man := FALSE;
   Fermi[1..6].Ctrl.Work_Man := FALSE;
   Fermi[1..6].Ctrl.Rest_Aut := FALSE;
   Fermi[1..6].Ctrl.Work_Aut := FALSE;
   Fermi[1..6].V.ValveCtrl.SafeStop := FALSE;
   Fermi[1..6].V.ValveCtrl.Rst := FALSE;
   Fermi[1..6].V.ValveCtrl.MoveRest := FALSE;
   Fermi[1..6].V.ValveCtrl.MoveWork := FALSE;
   Fermi[1..6].V.RestLimitSwitch := TRUE;
   Fermi[1..6].V.WorkLimitSwitch := FALSE;
   Fermi[1..6].V.OilInPressure := FALSE;
   Fermi[1..6].V.Simulation := FALSE;
   Fermi[1..6].V.Config.RestLimSwitchExist := TRUE;
   Fermi[1..6].V.Config.WorkLimSwitchExist := FALSE;
   Fermi[1..6].V.Config.CheckOilInPressure := FALSE;
   Fermi[1..6].V.Config.CutRestWhenIsAtRest := TRUE;
   Fermi[1..6].V.Config.CutWorkWhenIsAtWork := TRUE;
   Fermi[1..6].V.Config.RestTime := T#2S;
   Fermi[1..6].V.Config.WorkTime := T#2S;
   Fermi[1..6].V.Config.RestTimeOut := T#1H;
   Fermi[1..6].V.Config.WorkTimeOut := T#1H;
   Fermi[1..6].V.ValveSts.AlarmPresence := FALSE;
   Fermi[1..6].V.ValveSts.RestPermit := TRUE;
   Fermi[1..6].V.ValveSts.RestInProgress := FALSE;
   Fermi[1..6].V.ValveSts.IsAtRest := TRUE;
   Fermi[1..6].V.ValveSts.WorkPermit := TRUE;
   Fermi[1..6].V.ValveSts.WorkInProgress := FALSE;
   Fermi[1..6].V.ValveSts.IsAtWork := FALSE;
   Fermi[1..6].V.ValveSts.StandStill := TRUE;
   Fermi[1..6].V.RestSolenoid := FALSE;
   Fermi[1..6].V.WorkSolenoid := FALSE;
   Fermi[1..6].V.ReqOilPressure := FALSE;
   Fermi[1..6].V.IsAtRest := TRUE;
   Fermi[1..6].V.IsAtWork := FALSE;
   Fermi[1..6].V.Ctrl.RestReq := FALSE;
   Fermi[1..6].V.Ctrl.WorkReq := FALSE;
   Fermi[1..6].V.Ctrl.RestSolenoid := FALSE;
   Fermi[1..6].V.Ctrl.WorkSolenoid := FALSE;
   Fermi[1..6].V.tonRest.PT := T#2S;
   Fermi[1..6].V.tonRest.IN := TRUE;
   Fermi[1..6].V.tonWork.PT := T#0MS;
   Fermi[1..6].V.tonWork.IN := FALSE;
   Fermi[1..6].V.tonTimeOutRest.PT := T#0MS;
   Fermi[1..6].V.tonTimeOutRest.IN := FALSE;
   Fermi[1..6].V.tonTimeOutWork.PT := T#0MS;
   Fermi[1..6].V.tonTimeOutWork.IN := FALSE;
   Fermi[1..6].TON_NoPendingCmd.PT := T#500MS;
   Fermi[1..6].TON_NoPendingCmd.IN := TRUE;
   Fermi[1..6].TON_Rest_MissingExtEnable.PT := T#0MS;
   Fermi[1..6].TON_Rest_MissingExtEnable.IN := FALSE;
   Fermi[1..6].TON_Work_MissingExtEnable.PT := T#0MS;
   Fermi[1..6].TON_Work_MissingExtEnable.IN := FALSE;
   Fermi[1..6].TON_PressureRunning_Timeout.PT := T#0MS;
   Fermi[1..6].TON_PressureRunning_Timeout.IN := FALSE;
   Fermi[1..6].Aux.Pb_Rest := FALSE;
   Fermi[1..6].Aux.Pb_Work := FALSE;
   Fermi[1..6].Aux.Pb_StartStop := FALSE;
   TON_OP_REST_MissingCnd.PT := T#0MS;
   TON_OP_REST_MissingCnd.IN := FALSE;
   TON_OP_WORK_MissingCnd.PT := T#0MS;
   TON_OP_WORK_MissingCnd.IN := FALSE;
END_DATA_BLOCK

DATA_BLOCK "A0301_Ribaltatore"   // DB77
// stored: InstanceOfName A0301_Ribaltatore_FB, InstanceOfType FB
"A0301_Ribaltatore_FB"
BEGIN
END_DATA_BLOCK

DATA_BLOCK "A0301_Fermi_P4"   // DB46
// stored: InstanceOfName A0301_Fermi_P4_FB, InstanceOfType FB
"A0301_Fermi_P4_FB"
BEGIN
   HMI.Selection[1..6] := TRUE;
END_DATA_BLOCK

DATA_BLOCK "A0301_Spintore_Lat"   // DB121
// stored: InstanceOfName A0301_Spintore_Lat_FB, InstanceOfType FB
"A0301_Spintore_Lat_FB"
BEGIN
   HMI.Selection[1..6] := TRUE;
END_DATA_BLOCK

DATA_BLOCK "A0302_Manager"   // DB84
// stored: InstanceOfName A0302_Manager_FB, InstanceOfType FB
"A0302_Manager_FB"
BEGIN
END_DATA_BLOCK

DATA_BLOCK "A0302_Mng_BtrkListToCheck"   // DB182
// stored: InstanceOfName A0302_Mng_BtrkListToCheck_FB, InstanceOfType FB
"A0302_Mng_BtrkListToCheck_FB"
   // VAR_IN_OUT
   //    BTrk : Array[1.."BTRK_A03_EXIT_TOCHECK_ITEMS"] of "BTrk_item";
   //    FullList : Bool;
   // END_VAR
   // VAR
   //    i { ExternalAccessible := 'False'; ExternalVisible := 'False'; ExternalWritable := 'False'} : Int;
   //    j : Int;
   //    Control : Struct
   //       NoPlaceEmpty : USInt;
   //       StopCount : Bool;
   //       Pls_ClearArchive : Bool;
   //    END_STRUCT;
   // END_VAR
BEGIN
END_DATA_BLOCK

DATA_BLOCK "A0302_HU_Cytropack"   // DB81
// stored: InstanceOfName A0302_HU_Cytropack_FB, InstanceOfType FB
"A0302_HU_Cytropack_FB"
BEGIN
END_DATA_BLOCK

DATA_BLOCK "A0302_Spintore"   // DB109
// stored: InstanceOfName A0302_Spintore_FB, InstanceOfType FB
"A0302_Spintore_FB"
BEGIN
END_DATA_BLOCK

DATA_BLOCK "A0302_PareggiatoreCoda"   // DB152
// stored: InstanceOfName A0302_PareggiatoreCoda_FB, InstanceOfType FB
"A0302_PareggiatoreCoda_FB"
BEGIN
END_DATA_BLOCK

DATA_BLOCK "A0302_PareggiatoreTesta"   // DB122
// stored: InstanceOfName A0302_PareggiatoreTesta_FB, InstanceOfType FB
"A0302_PareggiatoreTesta_FB"
BEGIN
END_DATA_BLOCK

DATA_BLOCK "A0302_Manipolatore"   // DB117
// stored: InstanceOfName A0302_Manipolatore_FB, InstanceOfType FB
"A0302_Manipolatore_FB"
BEGIN
END_DATA_BLOCK

DATA_BLOCK "A0301_PTrk_To_BTrk_Create"   // DB183
// stored: InstanceOfName A0301_PTrk_To_BTrk_Create_FB, InstanceOfType FB
"A0301_PTrk_To_BTrk_Create_FB"
   // VAR_INPUT
   //    AreaInterface : "AreaInterface";
   //    Execute : Bool;
   //    PTrk_P2 { ExternalAccessible := 'False'; ExternalVisible := 'False'; ExternalWritable := 'False'} : "PTrk_Item";
   //    PTrk_P3 { ExternalAccessible := 'False'; ExternalVisible := 'False'; ExternalWritable := 'False'} : "PTrk_Item";
   // END_VAR
   // VAR_OUTPUT
   //    BTrk { ExternalAccessible := 'False'; ExternalVisible := 'False'; ExternalWritable := 'False'} : "BTrk_item";
   // END_VAR
   // VAR_IN_OUT
   //    Status : USInt;
   // END_VAR
   // VAR
   //    R_TRIG_Execute { S7_SetPoint := 'True'} : R_TRIG;
   //    Inc_Last_ID_B { ExternalAccessible := 'False'; ExternalVisible := 'False'; ExternalWritable := 'False'} : Bool;
   //    Alarm { ExternalAccessible := 'False'; ExternalVisible := 'False'; ExternalWritable := 'False'} : USInt;
   // END_VAR
BEGIN
END_DATA_BLOCK

DATA_BLOCK "Area0301_V_Counter_IDB"   // DB62
// stored: InstanceOfName VirtualEncoder, InstanceOfType FB
"VirtualEncoder"
   // VAR_INPUT
   //    ActualSpeed : LReal;
   //    OB_Cycle : UDInt;
   // END_VAR
   // VAR_IN_OUT
   //    VCounter : LReal;
   // END_VAR
   // VAR
   //    InitDone : Bool;
   //    ActualSpeed_mm_s : LReal;
   //    PrevSpeed_mm_s : LReal;
   //    DeltaT_s : LReal;
   //    DeltaV : LReal;
   //    DeltaS : LReal;
   // END_VAR
BEGIN
END_DATA_BLOCK

DATA_BLOCK "TIA_PN_FcP5020_DB"   // DB50153
// stored: InstanceOfName TIA_PN_FcP5020, InstanceOfType FB
"TIA_PN_FcP5020"
   // VAR_INPUT
   //    Enable : Bool;
   //    EnableDrive : Bool;
   //    ClearError : Bool;
   //    PressureCmd : Real;
   //    MaxSpeedLimit : Real;
   //    InputADDR : HW_IO;
   //    OutputADDR : HW_IO;
   // END_VAR
   // VAR_OUTPUT
   //    InOperation : Bool;
   //    MotorStarted : Bool;
   //    Error : Bool;
   //    Warning : Bool;
   //    DiagnosisCode : Word;
   //    Status : Word;
   //    PressureAct : Real;
   //    SpeedAct : Real;
   // END_VAR
   // VAR
   //    fbTON_TIME { S7_SetPoint := 'True'} : TON_TIME;
   //    bMbit0 : Bool;
   //    bMbit1 : Bool;
   //    bMbit2 : Bool;
   //    bMbit3 : Bool;
   //    bEnableRise : Bool;
   //    bErrorResetFall : Bool;
   //    bFBErrorFall : Bool;
   //    bClearErrorRise : Bool;
   //    stInputData { S7_SetPoint := 'True'} : "FCP_IN";
   //    stOutputData { S7_SetPoint := 'True'} : "FCP_OUT";
   //    hwInputADDR : HW_IO;
   //    hwOutputADDR : HW_IO;
   //    iStep : Int;
   //    iErrorStep : Int;
   //    iReturnVal : Int;
   //    wReturnVal : Word;
   //    bFBErrorPressureCmd : Bool;
   //    bFBErrorMaxSpeedLimit : Bool;
   //    bFBErrorDPRD_DPWR : Bool;
   //    bFcPError : Bool;
   //    bEFCError : Bool;
   //    bFcPWarning : Bool;
   //    bEFCWarning : Bool;
   //    rPressureCmdInternal : Real;
   //    rMaxSpeedLimtInternal : Real;
   //    bInternalRunTrigger : Bool;
   //    bInternalRun : Bool;
   // END_VAR
BEGIN
END_DATA_BLOCK

DATA_BLOCK "A0302_Bordatrice_RegolazioneFormato"   // DB74
// stored: InstanceOfName A0302_Bordatrice_RegolazioneFormato_FB, InstanceOfType FB
"A0302_Bordatrice_RegolazioneFormato_FB"
   // VAR_INPUT
   //    AreaInterface : "AreaInterface";
   //    ZSI : "udt_ZoneSafetyInterface";
   //    DSI_Formato : "udt_DeviceSafetyInterface";
   //    DSI_Cassetta : "udt_DeviceSafetyInterface";
   //    Cin : Struct
   //       LineSetup_Exe : Bool;
   //       OB30_High : Bool;
   //       Infeed_ON : Bool;
   //    END_STRUCT;
   //    DataIn : Struct
   //       PB_Passaggio01_Combo : "Ax_PB";
   //       PB_Passaggio02_Combo : "Ax_PB";
   //       PB_Passaggio03_Combo : "Ax_PB";
   //       PB_Passaggio04_Combo : "Ax_PB";
   //    END_STRUCT;
   // END_VAR
   // VAR_OUTPUT
   //    MachineInterface { ExternalAccessible := 'False'; ExternalVisible := 'False'; ExternalWritable := 'False'} : "MachineInterface";
   //    Cout : Struct
   //       OB30_High_Req : Bool;
   //       Infeed_ReqON : Bool;
   //       CtrlSafe_AX_M : Bool;
   //       SetUp_Bordatrice_Done : Array[1..9] of Bool;
   //    END_STRUCT;
   // END_VAR
   // VAR_IN_OUT
   //    Par_Machne : Struct
   //       Nervatura_Pos_Riposo : Real;
   //       Passaggio01_MaxDisallineamentoAXs : Real;
   //       Passaggio02_MaxDisallineamentoAXs : Real;
   //       Passaggio03_MaxDisallineamentoAXs : Real;
   //       Passaggio04_MaxDisallineamentoAXs : Real;
   //       AxD_AutoSpeed : Real;
   //    END_STRUCT;
   //    Par_Enc : Array[1..9] of "PosFbk_RTN";
   //    Par_D : Array[1..1] of "Positioning_DOL_Machine_Par";
   //    Par_M : Array[2..9] of "Positioning_MOL_Machine_Par";
   //    Pers_D : Array[1..1] of "Positioning_DOL_Machine_Pers_Data";
   //    Pers_M : Array[2..9] of "Positioning_MOL_Machine_Pers_Data";
   // END_VAR
   // VAR
   //    i : Int;
   //    Init_Done : Bool;
   //    HMI : Struct
   //       Passaggio01_Combo_TargetPos : Real;
   //       Passaggio02_Combo_TargetPos : Real;
   //       Passaggio03_Combo_TargetPos : Real;
   //       Passaggio04_Combo_TargetPos : Real;
   //    END_STRUCT;
   //    Warning : Struct
   //       Ax_D { S7_SetPoint := 'True'} : Array[1..1] of "Positioning_DOL_Machine_Wng";
   //       Ax_M : Array[1..9] of "Positioning_MOL_Machine_Wng";
   //       Passaggio01_MaxDisallineamentoAXs { S7_SetPoint := 'True'} : Bool;
   //       Passaggio02_MaxDisallineamentoAXs { S7_SetPoint := 'True'} : Bool;
   //       Passaggio03_MaxDisallineamentoAXs { S7_SetPoint := 'True'} : Bool;
   //       Passaggio04_MaxDisallineamentoAXs { S7_SetPoint := 'True'} : Bool;
   //    END_STRUCT;
   //    Alarm : Struct
   //       Enc : Array[1..9] of "PosFbk_Encoder_Alr";
   //       Ax_D { S7_SetPoint := 'True'} : Array[1..1] of "Positioning_DOL_Machine_Alr";
   //       Ax_M { S7_SetPoint := 'True'} : Array[1..9] of "Positioning_MOL_Machine_Alr";
   //    END_STRUCT;
   //    Sts : Struct
   //       UpdateSel : Int;
   //       Passaggio01 : Struct
   //          DeltaPos_OP_MOT : LReal;
   //          AxOP_Pause_Minus : Bool;
   //          AxOP_Pause_Plus : Bool;
   //          AxMOT_Pause_Minus : Bool;
   //          AxMOT_Pause_Plus : Bool;
   //       END_STRUCT;
   //       Passaggio02 : Struct
   //          DeltaPos_OP_MOT : LReal;
   //          AxOP_Pause_Minus : Bool;
   //          AxOP_Pause_Plus : Bool;
   //          AxMOT_Pause_Minus : Bool;
   //          AxMOT_Pause_Plus : Bool;
   //       END_STRUCT;
   //       Passaggio03 : Struct
   //          DeltaPos_OP_MOT : LReal;
   //          AxOP_Pause_Minus : Bool;
   //          AxOP_Pause_Plus : Bool;
   //          AxMOT_Pause_Minus : Bool;
   //          AxMOT_Pause_Plus : Bool;
   //       END_STRUCT;
   //       Passaggio04 : Struct
   //          DeltaPos_OP_MOT : LReal;
   //          AxOP_Pause_Minus : Bool;
   //          AxOP_Pause_Plus : Bool;
   //          AxMOT_Pause_Minus : Bool;
   //          AxMOT_Pause_Plus : Bool;
   //       END_STRUCT;
   //       TargetPos : Array[1..9] of Real;
   //    END_STRUCT;
   //    Ctrl : Struct
   //       OB30_High_Req : Bool;
   //       Passaggio01_Combo_MAN : Struct
   //          Minus : Bool;
   //          Plus : Bool;
   //          MoveToPos : Bool;
   //       END_STRUCT;
   //       Passaggio02_Combo_MAN : Struct
   //          Minus : Bool;
   //          Plus : Bool;
   //          MoveToPos : Bool;
   //       END_STRUCT;
   //       Passaggio03_Combo_MAN : Struct
   //          Minus : Bool;
   //          Plus : Bool;
   //          MoveToPos : Bool;
   //       END_STRUCT;
   //       Passaggio04_Combo_MAN : Struct
   //          Minus : Bool;
   //          Plus : Bool;
   //          MoveToPos : Bool;
   //       END_STRUCT;
   //    END_STRUCT;
   //    EncITF : Array[1..9] of "PosFbk_ITF";
   //    TOF_OB30_High { S7_SetPoint := 'True'} : TOF_TIME;
   //    Enc { S7_SetPoint := 'True'} : Array[1..9] of "PosFbk_SickAFM60";
   //    AX_D { S7_SetPoint := 'True'} : Array[1..1] of "Positioning_DOL_Machine_FB";
   //    AX_M { S7_SetPoint := 'True'} : Array[2..9] of "Positioning_MOL_Machine_FB";
   //    AUX : Struct
   //       PB_Passaggio01_Combo : Struct
   //          Minus : Bool;
   //          Plus : Bool;
   //          MoveToPos : Bool;
   //       END_STRUCT;
   //       PB_Passaggio02_Combo : Struct
   //          Minus : Bool;
   //          Plus : Bool;
   //          MoveToPos : Bool;
   //       END_STRUCT;
   //       PB_Passaggio03_Combo : Struct
   //          Minus : Bool;
   //          Plus : Bool;
   //          MoveToPos : Bool;
   //       END_STRUCT;
   //       PB_Passaggio04_Combo : Struct
   //          Minus : Bool;
   //          Plus : Bool;
   //          MoveToPos : Bool;
   //       END_STRUCT;
   //    END_STRUCT;
   // END_VAR
BEGIN
END_DATA_BLOCK

DATA_BLOCK "A0302_Bordatrice"   // DB92
// stored: InstanceOfName A0302_Bordatrice_FB, InstanceOfType FB
"A0302_Bordatrice_FB"
BEGIN
END_DATA_BLOCK

DATA_BLOCK "Lubr_Bordat_DB"   // DB227
// stored: InstanceOfName Lubr_Bordat, InstanceOfType FB
"Lubr_Bordat"
BEGIN
END_DATA_BLOCK

DATA_BLOCK "A0302_Rulliera"   // DB85
// stored: InstanceOfName A0302_Rulliera_FB, InstanceOfType FB
"A0302_Rulliera_FB"
BEGIN
END_DATA_BLOCK

DATA_BLOCK "A0302_Centratori"   // DB110
// stored: InstanceOfName A0302_Centratori_FB, InstanceOfType FB
"A0302_Centratori_FB"
BEGIN
   HMI.Selection.Centraggio[1..3] := TRUE;
   HMI.Selection.Sollevamento[1..3] := TRUE;
END_DATA_BLOCK
